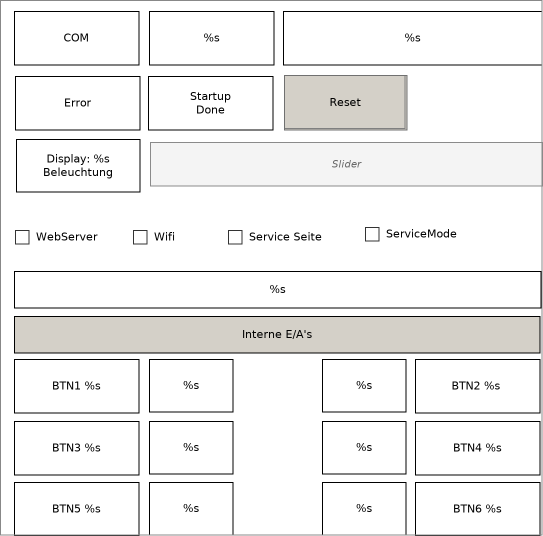
VISUALIZATION BusCYD6F_Frame  // 543x536
VAR_IN_OUT
	stBusTaster6F_Input		:ST_BusCYD6F_Input;
	stBusTaster6F_Output	:ST_BusTaster6F_Output;
	stBusTaster6F_Cnt		:ST_BusTaster6F_Cnt;
END_VAR
    Rectangle (14,11 125x54), "COM", colour toggle: stBusTaster6F_Output.bCOM
    Rectangle (14,359 125x54), "BTN1 %s", text variable: stBusTaster6F_Cnt.dwCntButtons[1], colour toggle: stBusTaster6F_Output.bButtons[1]
    Rectangle (149,11 125x54), "%s", text variable: stBusTaster6F_Input.diID
    Rectangle (283,11 259x54), "%s", text variable: stBusTaster6F_Input.sName
    Rectangle (415,359 125x54), "BTN2 %s", text variable: stBusTaster6F_Cnt.dwCntButtons[2], colour toggle: stBusTaster6F_Output.bButtons[2]
    Rectangle (14,421 125x54), "BTN3 %s", text variable: stBusTaster6F_Cnt.dwCntButtons[3], colour toggle: stBusTaster6F_Output.bButtons[3]
    Rectangle (415,421 125x54), "BTN4 %s", text variable: stBusTaster6F_Cnt.dwCntButtons[4], colour toggle: stBusTaster6F_Output.bButtons[4]
    Rectangle (14,482 125x54), "BTN5 %s", text variable: stBusTaster6F_Cnt.dwCntButtons[5], colour toggle: stBusTaster6F_Output.bButtons[5]
    Rectangle (415,482 125x54), "BTN6 %s", text variable: stBusTaster6F_Cnt.dwCntButtons[6], colour toggle: stBusTaster6F_Output.bButtons[6]
    Rectangle (149,359 84x53), "%s", text variable: stBusTaster6F_Input.iLED[1]
        OnMouseDown: write the text variable via VisuDialogs.Numpad, min 0, max 100
    Rectangle (322,359 84x53), "%s", text variable: stBusTaster6F_Input.iLED[2]
        OnMouseDown: write the text variable via VisuDialogs.Numpad, min 0, max 100
    Rectangle (149,421 84x53), "%s", text variable: stBusTaster6F_Input.iLED[3]
        OnMouseDown: write the text variable via VisuDialogs.Numpad, min 0, max 100
    Rectangle (322,421 84x53), "%s", text variable: stBusTaster6F_Input.iLED[4]
        OnMouseDown: write the text variable via VisuDialogs.Numpad, min 0, max 100
    Rectangle (149,482 84x53), "%s", text variable: stBusTaster6F_Input.iLED[5]
        OnMouseDown: write the text variable via VisuDialogs.Numpad, min 0, max 100
    Rectangle (322,482 84x53), "%s", text variable: stBusTaster6F_Input.iLED[6]
        OnMouseDown: write the text variable via VisuDialogs.Numpad, min 0, max 100
    Button (284,75 123x55), "Reset"
        tap stBusTaster6F_Input.bReset
    Rectangle (15,76 125x54), "Error", colour toggle: stBusTaster6F_Output.bError
    Rectangle (14,271 527x37), "%s", text variable: stBusTaster6F_Output.sState
    Rectangle (148,76 125x54), "Startup Done", colour toggle: stBusTaster6F_Output.bStartupDone
    Rectangle (16,139 124x53), "Display: %s Beleuchtung", text variable: stBusTaster6F_Input.iLEDBg
        OnMouseDown: write the text variable via VisuDialogs.Numpad, min 0, max 100
    Rectangle (14,316 526x37), "Interne E/A's"
    Slider (150,142 393x44), variable: stBusTaster6F_Input.iLEDBg, scale 0..100
    Checkbox (363,206 178x56), "ServiceMode", variable: stBusTaster6F_Input.bServiceMode
    Checkbox (13,213 121x48), "WebServer", variable: stBusTaster6F_Input.bWebServer, invisible if: not stBusTaster6F_Input.bServiceMode
    Checkbox (131,213 85x48), "Wifi", variable: stBusTaster6F_Input.bWifi, invisible if: not stBusTaster6F_Input.bServiceMode
    Checkbox (226,213 119x48), "Service Seite", variable: stBusTaster6F_Input.bService, invisible if: not stBusTaster6F_Input.bServiceMode
END_VISUALIZATION

(* stored: Version 1.1.0.1, ProductVersion 3.1.4024.12
   Visu BusCYD6F_Frame: Id {42f3f68d-ceeb-4980-81ba-76e4cc59bbb7} *)
